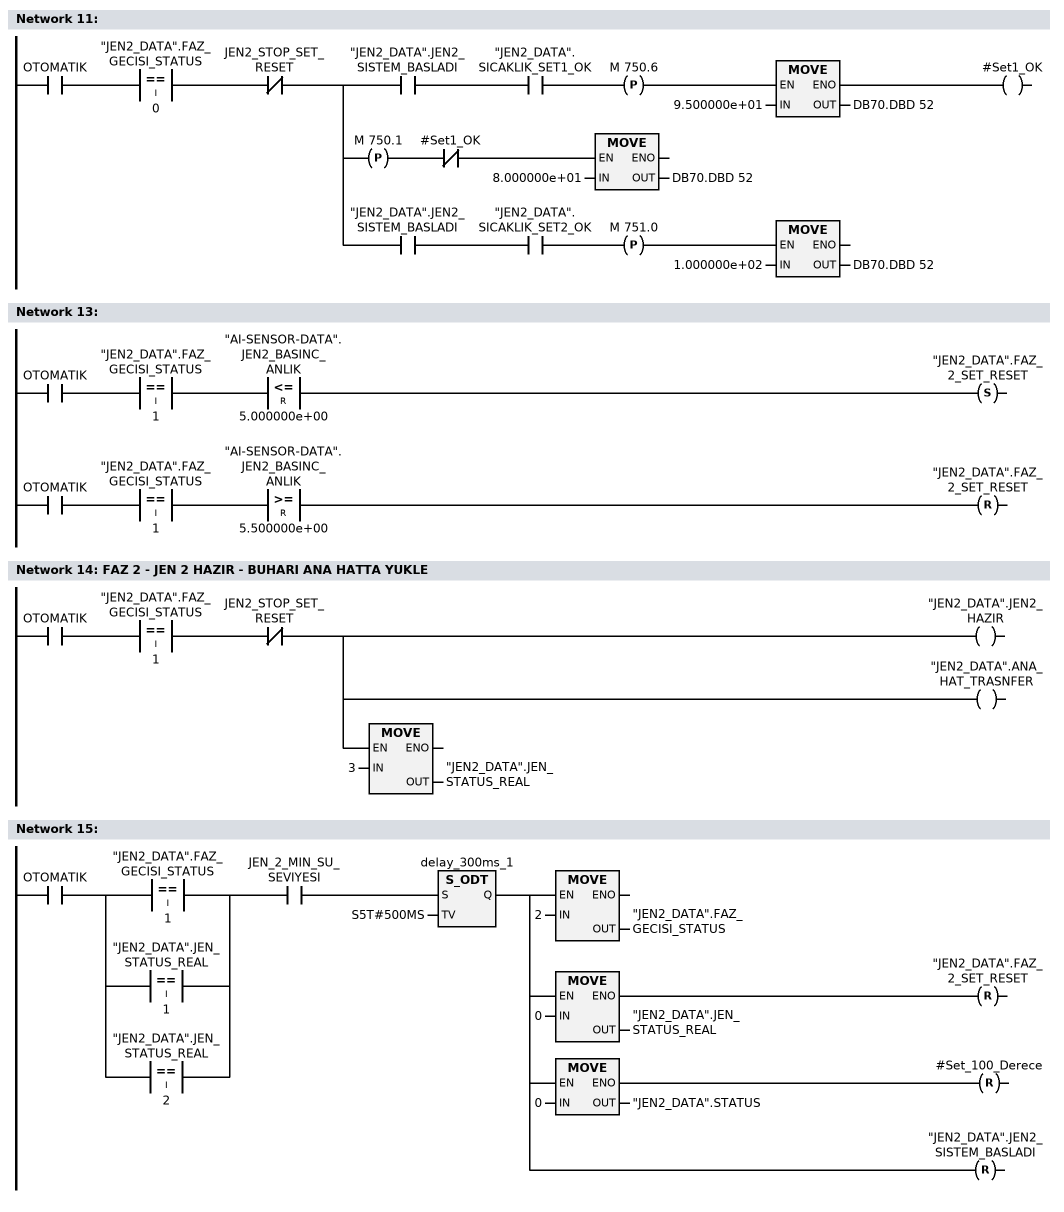
NETWORK
TITLE =
//-Sicaklik set 1 e geldiginde vana kapanma orani 5'e kadar düsüyor
//-Sicaklik set 2 e geldiginde vana kapanma orani 0'a kadar dusecek
      A     "OTOMATIK";
      A(;
      L     "JEN2_DATA".FAZ_GECISI_STATUS;
      L     0;
      ==I;
      );
      AN    "JEN2_STOP_SET_RESET";
      =     L 0.0;
      A     L 0.0;
      A     "JEN2_DATA".JEN2_SISTEM_BASLADI;
      A     "JEN2_DATA".SICAKLIK_SET1_OK;
      FP    M 750.6;
      JNB   _00c;
      L     9.500000e+01;
      T     DB70.DBD 52;
      SET;
      SAVE;
      CLR;
_00c: A     BR;
      =     #Set1_OK;
      A     L 0.0;
      FP    M 750.1;
      AN    #Set1_OK;
      JNB   _00d;
      L     8.000000e+01;
      T     DB70.DBD 52;
_00d: NOP   0;
      A     L 0.0;
      A     "JEN2_DATA".JEN2_SISTEM_BASLADI;
      A     "JEN2_DATA".SICAKLIK_SET2_OK;
      FP    M 751.0;
      JNB   _00e;
      L     1.000000e+02;
      T     DB70.DBD 52;
_00e: NOP   0;
NETWORK
TITLE =
NETWORK
TITLE =
//FAZ - 2 MODUNA GEÇ
//1-BURLOR VE POMPA 4.5-5.5 BAR ARASINDA ÇALISIP DURACAK
      A     "OTOMATIK";
      A(;
      L     "JEN2_DATA".FAZ_GECISI_STATUS;
      L     1;
      ==I;
      );
      A(;
      L     "AI-SENSOR-DATA".JEN2_BASINC_ANLIK;
      L     5.000000e+00;
      <=R;
      );
      S     "JEN2_DATA".FAZ_2_SET_RESET;
      A     "OTOMATIK";
      A(;
      L     "JEN2_DATA".FAZ_GECISI_STATUS;
      L     1;
      ==I;
      );
      A(;
      L     "AI-SENSOR-DATA".JEN2_BASINC_ANLIK;
      L     5.500000e+00;
      >=R;
      );
      R     "JEN2_DATA".FAZ_2_SET_RESET;
      NOP   0;
NETWORK
TITLE = FAZ 2 - JEN 2 HAZIR - BUHARI ANA HATTA YUKLE
      A     "OTOMATIK";
      A(;
      L     "JEN2_DATA".FAZ_GECISI_STATUS;
      L     1;
      ==I;
      );
      AN    "JEN2_STOP_SET_RESET";
      =     L 0.0;
      A     L 0.0;
      BLD   102;
      =     "JEN2_DATA".JEN2_HAZIR;
      A     L 0.0;
      BLD   102;
      =     "JEN2_DATA".ANA_HAT_TRASNFER;
      A     L 0.0;
      JNB   _00f;
      L     3;
      T     "JEN2_DATA".JEN_STATUS_REAL;
_00f: NOP   0;
NETWORK
TITLE =
//FAZ 3 - GUVENLIK ONLEMLERI 
//1- 6 bar asildiginda -ok
//2- Baca 180 dereceyi gecerse -ok
//3- Su miktari min altina duserse -ok
      A     "OTOMATIK";
      A(;
      O(;
      L     "JEN2_DATA".FAZ_GECISI_STATUS;
      L     1;
      ==I;
      );
      O(;
      L     "JEN2_DATA".JEN_STATUS_REAL;
      L     1;
      ==I;
      );
      O(;
      L     "JEN2_DATA".JEN_STATUS_REAL;
      L     2;
      ==I;
      );
      );
      A     "JEN_2_MIN_SU_SEVIYESI";
      L     S5T#500MS;
      SD    "delay_300ms_1";
      NOP   0;
      NOP   0;
      NOP   0;
      A     "delay_300ms_1";
      =     L 0.0;
      A     L 0.0;
      JNB   _010;
      L     2;
      T     "JEN2_DATA".FAZ_GECISI_STATUS;
_010: NOP   0;
      A     L 0.0;
      JNB   _011;
      L     0;
      T     "JEN2_DATA".JEN_STATUS_REAL;
      SET;
      SAVE;
      CLR;
_011: A     BR;
      R     "JEN2_DATA".FAZ_2_SET_RESET;
      A     L 0.0;
      JNB   _012;
      L     0;
      T     "JEN2_DATA".STATUS;
      SET;
      SAVE;
      CLR;
_012: A     BR;
      R     #Set_100_Derece;
      A     L 0.0;
      BLD   102;
      R     "JEN2_DATA".JEN2_SISTEM_BASLADI;
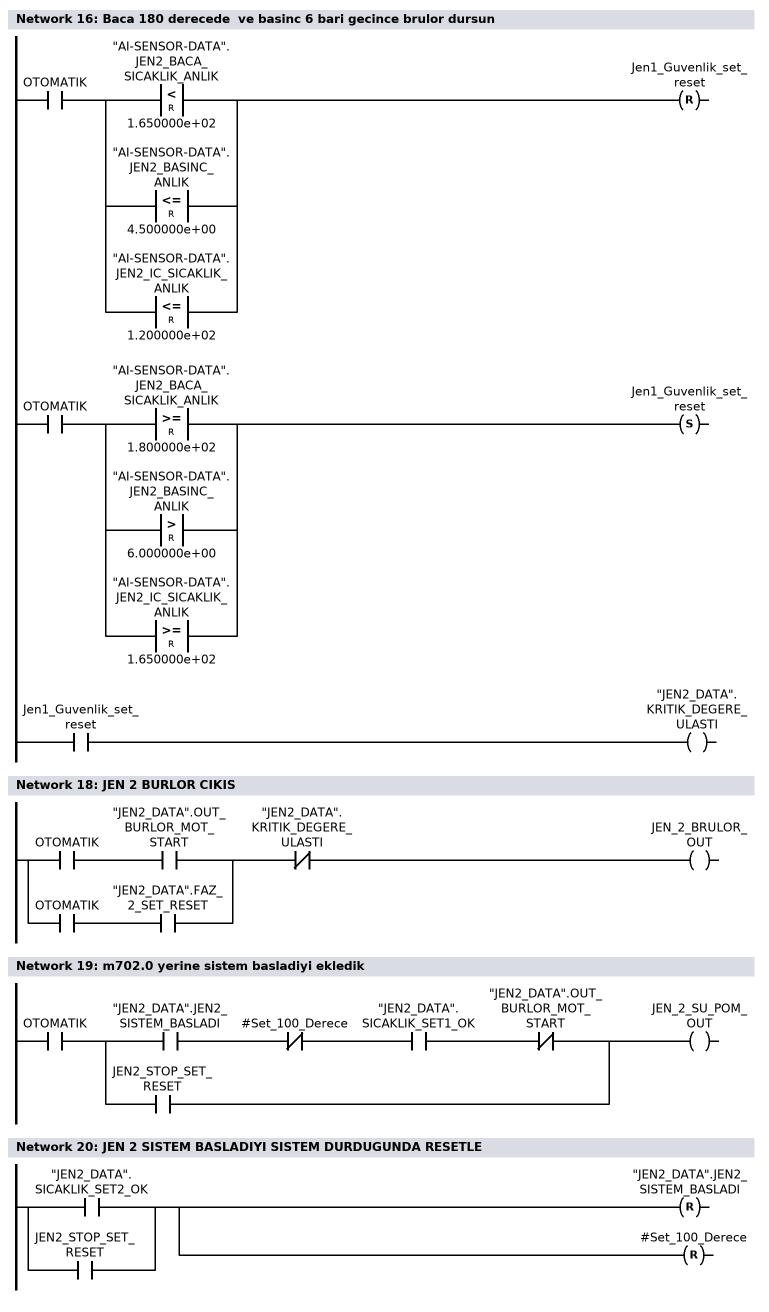
NETWORK
TITLE = Baca 180 derecede  ve basinc 6 bari gecince brulor dursun
      A     "OTOMATIK";
      A(;
      O(;
      L     "AI-SENSOR-DATA".JEN2_BACA_SICAKLIK_ANLIK;
      L     1.650000e+02;
      <R;
      );
      O(;
      L     "AI-SENSOR-DATA".JEN2_BASINC_ANLIK;
      L     4.500000e+00;
      <=R;
      );
      O(;
      L     "AI-SENSOR-DATA".JEN2_IC_SICAKLIK_ANLIK;
      L     1.200000e+02;
      <=R;
      );
      );
      R     "Jen1_Guvenlik_set_reset";
      A     "OTOMATIK";
      A(;
      O(;
      L     "AI-SENSOR-DATA".JEN2_BACA_SICAKLIK_ANLIK;
      L     1.800000e+02;
      >=R;
      );
      O(;
      L     "AI-SENSOR-DATA".JEN2_BASINC_ANLIK;
      L     6.000000e+00;
      >R;
      );
      O(;
      L     "AI-SENSOR-DATA".JEN2_IC_SICAKLIK_ANLIK;
      L     1.650000e+02;
      >=R;
      );
      );
      S     "Jen1_Guvenlik_set_reset";
      A     "Jen1_Guvenlik_set_reset";
      =     "JEN2_DATA".KRITIK_DEGERE_ULASTI;
NETWORK
TITLE =
NETWORK
TITLE = JEN 2 BURLOR CIKIS
      A(;
      A     "OTOMATIK";
      A     "JEN2_DATA".OUT_BURLOR_MOT_START;
      O;
      A     "OTOMATIK";
      A     "JEN2_DATA".FAZ_2_SET_RESET;
      );
      AN    "JEN2_DATA".KRITIK_DEGERE_ULASTI;
      =     "JEN_2_BRULOR_OUT";
NETWORK
TITLE = m702.0 yerine sistem basladiyi ekledik
      A     "OTOMATIK";
      A(;
      A     "JEN2_DATA".JEN2_SISTEM_BASLADI;
      AN    #Set_100_Derece;
      A     "JEN2_DATA".SICAKLIK_SET1_OK;
      AN    "JEN2_DATA".OUT_BURLOR_MOT_START;
      O     "JEN2_STOP_SET_RESET";
      );
      =     "JEN_2_SU_POM_OUT";
NETWORK
TITLE = JEN 2 SISTEM BASLADIYI SISTEM DURDUGUNDA RESETLE
      O     "JEN2_DATA".SICAKLIK_SET2_OK;
      O     "JEN2_STOP_SET_RESET";
      R     "JEN2_DATA".JEN2_SISTEM_BASLADI;
      R     #Set_100_Derece;
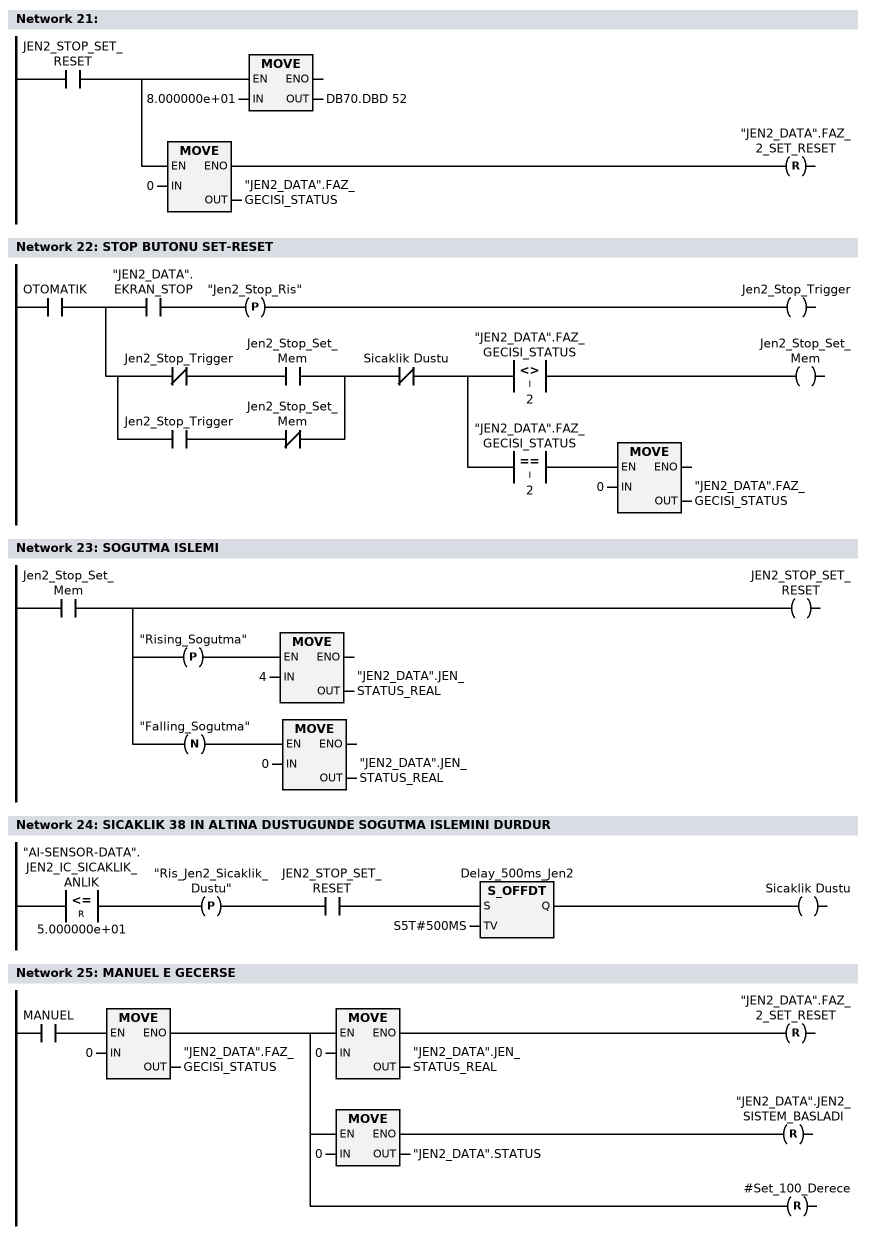
NETWORK
TITLE =
      A     "JEN2_STOP_SET_RESET";
      =     L 0.0;
      A     L 0.0;
      JNB   _013;
      L     8.000000e+01;
      T     DB70.DBD 52;
_013: NOP   0;
      A     L 0.0;
      JNB   _014;
      L     0;
      T     "JEN2_DATA".FAZ_GECISI_STATUS;
      SET;
      SAVE;
      CLR;
_014: A     BR;
      R     "JEN2_DATA".FAZ_2_SET_RESET;
NETWORK
TITLE = STOP BUTONU SET-RESET
      A     "OTOMATIK";
      =     L 0.0;
      A     L 0.0;
      A     "JEN2_DATA".EKRAN_STOP;
      FP    "Jen2_Stop_Ris";
      =     "Jen2_Stop_Trigger";
      A     L 0.0;
      A(;
      AN    "Jen2_Stop_Trigger";
      A     "Jen2_Stop_Set_Mem";
      O;
      A     "Jen2_Stop_Trigger";
      AN    "Jen2_Stop_Set_Mem";
      );
      AN    "Sicaklik Dustu";
      =     L 0.1;
      A     L 0.1;
      A(;
      L     "JEN2_DATA".FAZ_GECISI_STATUS;
      L     2;
      <>I;
      );
      =     "Jen2_Stop_Set_Mem";
      A     L 0.1;
      A(;
      L     "JEN2_DATA".FAZ_GECISI_STATUS;
      L     2;
      ==I;
      );
      JNB   _015;
      L     0;
      T     "JEN2_DATA".FAZ_GECISI_STATUS;
_015: NOP   0;
NETWORK
TITLE = SOGUTMA ISLEMI
      A     "Jen2_Stop_Set_Mem";
      =     L 0.0;
      A     L 0.0;
      BLD   102;
      =     "JEN2_STOP_SET_RESET";
      A     L 0.0;
      FP    "Rising_Sogutma";
      JNB   _016;
      L     4;
      T     "JEN2_DATA".JEN_STATUS_REAL;
_016: NOP   0;
      A     L 0.0;
      FN    "Falling_Sogutma";
      JNB   _017;
      L     0;
      T     "JEN2_DATA".JEN_STATUS_REAL;
_017: NOP   0;
NETWORK
TITLE = SICAKLIK 38 IN ALTINA DUSTUGUNDE SOGUTMA ISLEMINI DURDUR
      A(;
      L     "AI-SENSOR-DATA".JEN2_IC_SICAKLIK_ANLIK;
      L     5.000000e+01;
      <=R;
      );
      FP    "Ris_Jen2_Sicaklik_Dustu";
      A     "JEN2_STOP_SET_RESET";
      L     S5T#500MS;
      SF    "Delay_500ms_Jen2";
      NOP   0;
      NOP   0;
      NOP   0;
      A     "Delay_500ms_Jen2";
      =     "Sicaklik Dustu";
NETWORK
TITLE = MANUEL E GECERSE
      A     "MANUEL";
      JNB   _018;
      L     0;
      T     "JEN2_DATA".FAZ_GECISI_STATUS;
      SET;
      SAVE;
      CLR;
_018: A     BR;
      =     L 0.0;
      A     L 0.0;
      JNB   _019;
      L     0;
      T     "JEN2_DATA".JEN_STATUS_REAL;
      SET;
      SAVE;
      CLR;
_019: A     BR;
      R     "JEN2_DATA".FAZ_2_SET_RESET;
      A     L 0.0;
      JNB   _01a;
      L     0;
      T     "JEN2_DATA".STATUS;
      SET;
      SAVE;
      CLR;
_01a: A     BR;
      R     "JEN2_DATA".JEN2_SISTEM_BASLADI;
      A     L 0.0;
      BLD   102;
      R     #Set_100_Derece;
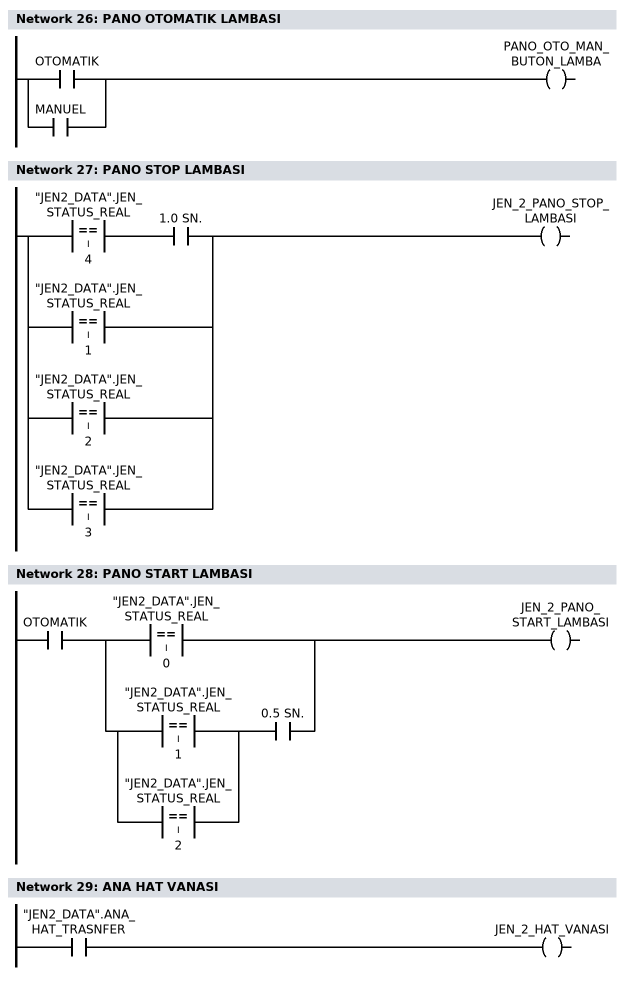
NETWORK
TITLE = PANO OTOMATIK LAMBASI
      O     "OTOMATIK";
      O     "MANUEL";
      =     "PANO_OTO_MAN_BUTON_LAMBA";
NETWORK
TITLE = PANO STOP LAMBASI
//1- Buhar hazýrlaniyor
//2- set 1 e ulasti
//3- Basinci Stabil tutma
//4- Sogutma
      A(;
      L     "JEN2_DATA".JEN_STATUS_REAL;
      L     4;
      ==I;
      );
      A     "1.0 SN.";
      O(;
      L     "JEN2_DATA".JEN_STATUS_REAL;
      L     1;
      ==I;
      );
      O(;
      L     "JEN2_DATA".JEN_STATUS_REAL;
      L     2;
      ==I;
      );
      O(;
      L     "JEN2_DATA".JEN_STATUS_REAL;
      L     3;
      ==I;
      );
      =     "JEN_2_PANO_STOP_LAMBASI";
NETWORK
TITLE = PANO START LAMBASI
      A     "OTOMATIK";
      A(;
      O(;
      L     "JEN2_DATA".JEN_STATUS_REAL;
      L     0;
      ==I;
      );
      O;
      A(;
      O(;
      L     "JEN2_DATA".JEN_STATUS_REAL;
      L     1;
      ==I;
      );
      O(;
      L     "JEN2_DATA".JEN_STATUS_REAL;
      L     2;
      ==I;
      );
      );
      A     "0.5 SN.";
      );
      =     "JEN_2_PANO_START_LAMBASI";
NETWORK
TITLE = ANA HAT VANASI 
      A     "JEN2_DATA".ANA_HAT_TRASNFER;
      =     "JEN_2_HAT_VANASI";
END_FUNCTION_BLOCK

FUNCTION "TIME_UNSCALE" : VOID	// FC 1
VERSION : 0.0
VAR_INPUT
  iTimeET : TIME ;
  iIstenileSure : S5TIME ;
END_VAR
VAR_OUTPUT
  oOUT : DINT ;
END_VAR
VAR_TEMP
  vTemp : DINT ;
  vValue : DINT ;
  vValue2 : DINT ;
  vIstenilenTime : TIME ;
  vIstenilenDint : DINT ;
END_VAR
BEGIN
// body was compiled from an SCL source; compiled code not shown
END_FUNCTION

// FC 33: know-how protected block, not included

// FC 105: know-how protected block, not included

// FC 106: know-how protected block, not included

DATA_BLOCK "AI-SENSOR-DATA"	// DB 1
VERSION : 0.1
  STRUCT
   JEN1_BASINC_ANLIK : REAL ;
   JEN2_BASINC_ANLIK : REAL ;
   JEN1_BASINC_RET_VAL : WORD ;
   JEN2_BASINC_RET_VAL : WORD ;
   JEN1_IC_SICAKLIK_ANLIK : REAL ;
   JEN2_IC_SICAKLIK_ANLIK : REAL ;
   JEN1_IC_SICAKLIK_RET_VAL : WORD ;
   JEN2_IC_SICAKLIK_RET_VAL : WORD ;
   JEN1_BACA_SICAKLIK_ANLIK : REAL ;
   JEN2_BACA_SICAKLIK_ANLIK : REAL ;
   JEN1_BACA_SICAKLIK_RET_V : WORD ;
   JEN2_BACA_SICAKLIK_RET_V : WORD ;
   HAT_BASINCI_RET_V : WORD ;
   HAT_BASINCI_ANLIK : REAL ;
   HAVA_BASINCI_RET_V : WORD ;
   HAVA_BASINCI_ANLIK : REAL ;
   HAT_BASINCI_YETERLI : BOOL ;
  END_STRUCT ;	
BEGIN
END_DATA_BLOCK

DATA_BLOCK "ORTAK_DATA"	// DB 2
VERSION : 0.1
  STRUCT
   JEN_EMNIYET_BASINCI : REAL ;
   JEN_EMNIYET_SICAKLIGI : REAL ;
   OTO_EMNIYET_BASINCI : REAL ;
   OTO_EMNIYET_SICAKLIGI : REAL ;
   OTO_ISLEM_BITTI_VANA_AC : BOOL ;
   OTO_JEN_DURDU : REAL ;
  END_STRUCT ;	
BEGIN
END_DATA_BLOCK

DATA_BLOCK "TIME_OTO_1_DB"	// DB 5
AUTHOR : SIMATIC
FAMILY : IEC_TC
VERSION : 0.0
"TON"
BEGIN
END_DATA_BLOCK

DATA_BLOCK "TIME_OTO_2_DB"	// DB 6
AUTHOR : SIMATIC
FAMILY : IEC_TC
VERSION : 0.0
"TON"
BEGIN
END_DATA_BLOCK

DATA_BLOCK "TIME_OTO_1_PROSES_DB"	// DB 7
AUTHOR : SIMATIC
FAMILY : IEC_TC
VERSION : 0.0
"TON"
BEGIN
END_DATA_BLOCK

DATA_BLOCK "TIME_OTO_2_PROSES_DB"	// DB 8
AUTHOR : SIMATIC
FAMILY : IEC_TC
VERSION : 0.0
"TON"
BEGIN
END_DATA_BLOCK

DATA_BLOCK DB 9
AUTHOR : SIMATIC
FAMILY : IEC_TC
VERSION : 0.0
"TON"
BEGIN
END_DATA_BLOCK

DATA_BLOCK DB 10
AUTHOR : SIMATIC
FAMILY : IEC_TC
VERSION : 0.0
"TON"
BEGIN
END_DATA_BLOCK

DATA_BLOCK "SURELER_DB"	// DB 14
VERSION : 0.0
"SURELER"
BEGIN
END_DATA_BLOCK

DATA_BLOCK "SAFETY_DB"	// DB 15
VERSION : 0.0
"SAFETY"
BEGIN
END_DATA_BLOCK

DATA_BLOCK "KAZAN1_DATA"	// DB 17
VERSION : 0.1
  STRUCT
   IN_STATUS : INT ;
   IN_JEN_OK : BOOL ;
   IN_DIGER_KAZ_TRANS_HAZIR : BOOL ;
   IN_PISIM_SURESI : S5TIME ;
   IN_SCALE_BASINC_PER : INT ;
   IN_SET_BASINC : REAL ;
   IN_DIGER_KAZAN_BASINCI : REAL ;
   O_PID_MAN_ON : BOOL ;
   O_PID_MAN : REAL ;
   O_TRANSFER_YAPILIYOR : BOOL ;
   O_SCALE_BASINC_RET_VAL : WORD ;
   O_SCALE_BASINC_OUT : REAL ;
   O_TRANSFERE_HAZIR : BOOL ;
   O_SCALE_SICAKLIK_RET_VAL : WORD ;
   O_SCALE_SICAKLIK_OUT : REAL ;
   IN_SCALE_SICAKLIK_PER : INT ;
   O_KAZAN_BOSALTIMDA : BOOL ;
   IN_DIGER_KAZ_BOSALTIMDA : BOOL ;
   IN_DIGER_KAZ_TRANSFERDE : BOOL ;
   O_PISIM_BASLADI : BOOL ;
   PISIM_GECEN_SURE_TIME : TIME ;
   PISIM_GECEN_SURE_DINT : DINT ;
   PROSES_SURESI_TIME : TIME ;
   PROSES_SURESI_DINT : DINT ;
   BEKLEME_SURESI_TIME : TIME ;
   BEKLEME_SURESI_DINT : DINT ;
  END_STRUCT ;	
BEGIN
END_DATA_BLOCK

DATA_BLOCK "KAZAN2_DATA"	// DB 18
VERSION : 0.1
  STRUCT
   IN_STATUS : INT ;
   IN_JEN_OK : BOOL ;
   IN_DIGER_KAZ_TRANS_HAZIR : BOOL ;
   IN_PISIM_SURESI : S5TIME ;
   IN_SCALE_BASINC_PER : INT ;
   IN_SET_BASINC : REAL ;
   IN_DIGER_KAZAN_BASINCI : REAL ;
   O_PID_MAN_ON : BOOL ;
   O_PID_MAN : REAL ;
   O_TRANSFER_YAPILIYOR : BOOL ;
   O_SCALE_BASINC_RET_VAL : WORD ;
   O_SCALE_BASINC_OUT : REAL ;
   O_TRANSFERE_HAZIR : BOOL ;
   O_SCALE_SICAKLIK_RET_VAL : WORD ;
   O_SCALE_SICAKLIK_OUT : REAL ;
   IN_SCALE_SICAKLIK_PER : INT ;
   O_KAZAN_BOSALTIMDA : BOOL ;
   IN_DIGER_KAZ_BOSALTIMDA : BOOL ;
   IN_DIGER_KAZ_TRANSFERDE : BOOL ;
   O_PISIM_BASLADI : BOOL ;
   PISIM_GECEN_SURE_TIME : TIME ;
   PISIM_GECEN_SURE_DINT : DINT ;
   PROSES_SURESI_TIM : TIME ;
   PROSES_SURESI_DINT : DINT ;
   BEKLEME_SURESI_TIME : TIME ;
   BEKLEME_SURESI_DINT : DINT ;
  END_STRUCT ;	
BEGIN
END_DATA_BLOCK

DATA_BLOCK "JEN1_DATA"	// DB 19
VERSION : 0.1
  STRUCT
   BASINC_SET_POINT : REAL ;
   STATUS : INT ;
   SICAKLIK_SET_POINT_1 : REAL ;
   SICAKLIK_SET_POINT_2 : REAL ;
   SISTEM_BASLADI : BOOL ;
   EKRAN_START : BOOL ;
   EKRAN_STOP : BOOL ;
   OUT_BURLOR_MOT_START : BOOL ;
   SICAKLIK_SET1_OK : BOOL ;
   SICAKLIK_SET2_OK : BOOL ;
   OUT_PID_START : BOOL ;
   FAZ_GECISI_STATUS : INT ;
   FAZ_2_SET_RESET : BOOL ;
   BAR_5_E_ULASTI : BOOL ;
   JEN1_HAZIR : BOOL ;
   ANA_HAT_TRASFER_HAZIR : BOOL ;
   JEN_STATUS_REAL : INT ;
   STOP_SET_RESET : BOOL ;
   CALISMA_SURESI_TIME : TIME ;
   CALISMA_SURESI_DINT : DINT ;
   KRITIK_DEGERLERE_ULASTI : BOOL ;	//180 derece baca-6 bari gecti- 165 ic sicaklik
   CALISMA_SURESI_EKRAN : DINT ;
   SET2_DEGERINE_ULASMADI : BOOL ;
  END_STRUCT ;	
BEGIN
END_DATA_BLOCK

DATA_BLOCK "JEN2_DATA"	// DB 20
VERSION : 0.1
  STRUCT
   BASINC_SET_POINT : REAL ;
   STATUS : INT ;
   SICAKLIK_SET_POINT_1 : REAL ;
   SICAKLIK_SET_POINT_2 : REAL ;
   JEN2_SISTEM_BASLADI : BOOL ;
   EKRAN_START : BOOL ;
   EKRAN_STOP : BOOL ;
   OUT_BURLOR_MOT_START : BOOL ;
   SICAKLIK_SET1_OK : BOOL ;
   SICAKLIK_SET2_OK : BOOL ;
   OUT_PID_START : BOOL ;
   FAZ_GECISI_STATUS : INT ;
   FAZ_2_SET_RESET : BOOL ;
   BAR_5_E_ULASTI : BOOL ;
   JEN2_HAZIR : BOOL ;
   ANA_HAT_TRASNFER : BOOL ;
   JEN_STATUS_REAL : INT ;
   STOP_SET_RESET : BOOL ;
   CALISMA_SURESI_TIME : TIME ;
   CALISMA_SURESI_DINT : DINT ;
   KRITIK_DEGERE_ULASTI : BOOL ;	//Baca 180 derecede-6 bari gecti-165 ic sicaklik
   CALISMA_SURESI_EKRAN : DINT ;
  END_STRUCT ;	
BEGIN
END_DATA_BLOCK

DATA_BLOCK "JEN1_PID_DATA"	// DB 21
VERSION : 0.1
  STRUCT
   TCONT_C_LMN : REAL ;
   TCONT_C_LMN_PER : INT ;
  END_STRUCT ;	
BEGIN
END_DATA_BLOCK

DATA_BLOCK "JEN2_PID_DATA"	// DB 22
VERSION : 0.1
  STRUCT
   TCONT_C_LMN : REAL ;
   TCONT_C_LMN_PER : INT ;
  END_STRUCT ;	
BEGIN
END_DATA_BLOCK

DATA_BLOCK "KAZAN1_PID_DATA"	// DB 23
VERSION : 0.1
  STRUCT
   TCONT_LMN_PER : INT ;
   TCONT_LMN : REAL ;
  END_STRUCT ;	
BEGIN
END_DATA_BLOCK

DATA_BLOCK "KAZAN2_PID_DATA"	// DB 24
VERSION : 0.1
  STRUCT
   TCONT_LMN_PER : INT ;
   TCONT_LMN : REAL ;
  END_STRUCT ;	
BEGIN
END_DATA_BLOCK

DATA_BLOCK DB 50
AUTHOR : SIMATIC
FAMILY : ICONT
VERSION : 0.0
"CONT_C"
BEGIN
END_DATA_BLOCK

DATA_BLOCK "JEN2_KONTROL_BLOGU_DB"	// DB 51
VERSION : 0.0
"JEN2_PID_KONTROL"
BEGIN
END_DATA_BLOCK

DATA_BLOCK DB 52
VERSION : 0.0
"JEN1_PID_KONTROL"
BEGIN
END_DATA_BLOCK

DATA_BLOCK "JEN_1_PID_DB"	// DB 69
AUTHOR : SIMATIC
FAMILY : CONTROL
VERSION : 0.0
"TCONT_CP"
BEGIN
END_DATA_BLOCK

DATA_BLOCK "JEN_2_PID_DB"	// DB 70
AUTHOR : SIMATIC
FAMILY : CONTROL
VERSION : 0.0
"TCONT_CP"
BEGIN
END_DATA_BLOCK

DATA_BLOCK "OTOKLAV_1_DB"	// DB 94
VERSION : 0.0
"KAZAN_1_KONTROL"
BEGIN
END_DATA_BLOCK

DATA_BLOCK "OTOKLAV_2_DB"	// DB 95
VERSION : 0.0
"KAZAN_2_KONTROL"
BEGIN
END_DATA_BLOCK

DATA_BLOCK "FB98_DB"	// DB 98
VERSION : 0.0
"JEN1_KONTROL_BLOGU"
BEGIN
END_DATA_BLOCK

DATA_BLOCK "FB99_DB"	// DB 99
VERSION : 0.0
"JEN2_KONTROL_BLOGU"
BEGIN
END_DATA_BLOCK

DATA_BLOCK DB 120
VERSION : 0.0
"KAZAN_ORTAK"
BEGIN
END_DATA_BLOCK

DATA_BLOCK "KAZAN_1_PID_DB"	// DB 130
AUTHOR : SIMATIC
FAMILY : CONTROL
VERSION : 0.0
"TCONT_CP"
BEGIN
END_DATA_BLOCK

DATA_BLOCK DB 131
VERSION : 0.0
"KAZAN_1_PID_KONTROL"
BEGIN
END_DATA_BLOCK

DATA_BLOCK DB 132
VERSION : 0.0
"KAZAN_2_PID_KONTROL"
BEGIN
END_DATA_BLOCK

DATA_BLOCK DB 230
VERSION : 0.0
"KAZAN_ORTAK"
BEGIN
END_DATA_BLOCK

DATA_BLOCK "KAZAN_2_PID_DATA"	// DB 231
AUTHOR : SIMATIC
FAMILY : CONTROL
VERSION : 0.0
"TCONT_CP"
BEGIN
END_DATA_BLOCK

DATA_BLOCK DB 232
VERSION : 0.0
"TEST_BLOGU"
BEGIN
END_DATA_BLOCK

ORGANIZATION_BLOCK OB 1
TITLE = "Main Program Sweep (Cycle)"
VERSION : 0.1
VAR_TEMP
  OB1_EV_CLASS : BYTE ;	//Bits 0-3 = 1 (Coming event), Bits 4-7 = 1 (Event class 1)
  OB1_SCAN_1 : BYTE ;	//1 (Cold restart scan 1 of OB 1), 3 (Scan 2-n of OB 1)
  OB1_PRIORITY : BYTE ;	//Priority of OB Execution
  OB1_OB_NUMBR : BYTE ;	//1 (Organization block 1, OB1)
  OB1_RESERVED_1 : BYTE ;	//Reserved for system
  OB1_RESERVED_2 : BYTE ;	//Reserved for system
  OB1_PREV_CYCLE : INT ;	//Cycle time of previous OB1 scan (milliseconds)
  OB1_MIN_CYCLE : INT ;	//Minimum cycle time of OB1 (milliseconds)
  OB1_MAX_CYCLE : INT ;	//Maximum cycle time of OB1 (milliseconds)
  OB1_DATE_TIME : DATE_AND_TIME ;	//Date and time OB1 started
END_VAR
BEGIN
NETWORK
TITLE = ALWAYS OFF
      UC    "MAINBLOCK";
NETWORK
TITLE = HAVA VE HAT BASINCI
      CALL  "SCALE" (
           $1                       := P#P 292.0,
           $2                       := L#1092616192,
           $3                       := L#0,
           $4                       := "ALWAYS OFF",
           $5                       := "AI-SENSOR-DATA".HAT_BASINCI_RET_V,
           $6                       := "AI-SENSOR-DATA".HAT_BASINCI_ANLIK);
      CALL  "SCALE" (
           $1                       := P#P 294.0,
           $2                       := L#1092616192,
           $3                       := L#0,
           $4                       := "ALWAYS OFF",
           $5                       := "AI-SENSOR-DATA".HAVA_BASINCI_RET_V,
           $6                       := "AI-SENSOR-DATA".HAVA_BASINCI_ANLIK);
NETWORK
TITLE = ACIKLAMALAR
//FB98 - JEN 1 KONTROL BLOGU
//FB99 - JEN 2 KONTROL BLOGU
//FB49 - JEN 1 PID KONTROL - PID BLOKLARI
//FB50 - JEN 2 PID KONTROL - PID BLOKLARI
//FB94 - KAZAN 1 KONTROL BLOGU - KAZAN 1 ILE ILGILI KONTROLLER
//FB95 - KAZAN 2 KONTROL BLOGU - KAZAN 2 ILE ILGILI KONTROLLER
//FB47 - KAZAN 1 PID KONTROL
//FB48 - KAZAN 2 PID KONTROL
//FB3 - SURELER - KAZAN1,KAZAN2, JEN1, JEN2 ILE ILGILI TUM SURELER BURADA TUTULUR
//FB2 - SAFETY
//      1)JEN1, JEN2 KRITIK SU SEVIYE MIKTARLARI
//      2)HAVA BASINCI KONTROLU
//      3)JENERATOR IS BITIMINDE BORUDA KALAN BUHARIN TAHLIYESI
//FB1 - MAINBLOCK  
//      1)ÇALISACAK TUM BLOKLAR BURADA CAGRILIR
//      2)AYRICA HAVA VE HAT BASINCI DONUSUMLARI BURADADIR
//FB5 - TEST BLOGU - PROSESIN DEVREYE ALINAMADAN ONCEKI TEST ISLEMLERININ GERCEKLESTIGI
//      BLOKTUR.
END_ORGANIZATION_BLOCK

ORGANIZATION_BLOCK "PID BLOCK"	// OB 35
TITLE = "Cyclic Interrupt"
VERSION : 0.1
VAR_TEMP
  OB35_EV_CLASS : BYTE ;	//Bits 0-3 = 1 (Coming event), Bits 4-7 = 1 (Event class 1)
  OB35_STRT_INF : BYTE ;	//16#36 (OB 35 has started)
  OB35_PRIORITY : BYTE ;	//Priority of OB Execution
  OB35_OB_NUMBR : BYTE ;	//35 (Organization block 35, OB35)
  OB35_RESERVED_1 : BYTE ;	//Reserved for system
  OB35_RESERVED_2 : BYTE ;	//Reserved for system
  OB35_PHASE_OFFSET : WORD ;	//Phase offset (msec)
  OB35_RESERVED_3 : INT ;	//Reserved for system
  OB35_EXC_FREQ : INT ;	//Frequency of execution (msec)
  OB35_DATE_TIME : DATE_AND_TIME ;	//Date and time OB35 started
END_VAR
BEGIN
NETWORK
TITLE =
      CALL  "JEN1_PID_KONTROL" , DB 52;
      CALL  "JEN2_PID_KONTROL" , "JEN2_KONTROL_BLOGU_DB";
NETWORK
TITLE =
      CALL  "KAZAN_1_PID_KONTROL" , DB 131;
      CALL  "KAZAN_2_PID_KONTROL" , DB 132;
END_ORGANIZATION_BLOCK

ORGANIZATION_BLOCK "ZAMANHATASI"	// OB 80
TITLE = "Cycle Time Fault"
VERSION : 0.1
VAR_TEMP
  OB80_EV_CLASS : BYTE ;	//16#35, Event class 3, Entering event state, Internal fault event
  OB80_FLT_ID : BYTE ;	//16#XX, Fault identifcation code
  OB80_PRIORITY : BYTE ;	//Priority of OB Execution
  OB80_OB_NUMBR : BYTE ;	//80 (Organization block 80, OB80)
  OB80_RESERVED_1 : BYTE ;	//Reserved for system
  OB80_RESERVED_2 : BYTE ;	//Reserved for system
  OB80_ERROR_INFO : WORD ;	//Error information on event
  OB80_ERR_EV_CLASS : BYTE ;	//Class of event causing error
  OB80_ERR_EV_NUM : BYTE ;	//Number of event causing error
  OB80_OB_PRIORITY : BYTE ;	//Priority of OB causing error
  OB80_OB_NUM : BYTE ;	//Number of OB causing error
  OB80_DATE_TIME : DATE_AND_TIME ;	//Date and time OB80 started
END_VAR
BEGIN
// (block stored without names or comments; labels and parameter names are numbered)
END_ORGANIZATION_BLOCK

ORGANIZATION_BLOCK "GERILIMHATASI"	// OB 81
TITLE = "Power Supply Fault"
VERSION : 0.1
VAR_TEMP
  OB81_EV_CLASS : BYTE ;	//16#39, Event class 3, Entering event state, Internal fault event
  OB81_FLT_ID : BYTE ;	//16#XX, Fault identifcation code
  OB81_PRIORITY : BYTE ;	//Priority of OB Execution
  OB81_OB_NUMBR : BYTE ;	//81 (Organization block 81, OB81)
  OB81_RESERVED_1 : BYTE ;	//Reserved for system
  OB81_RESERVED_2 : BYTE ;	//Reserved for system
  OB81_RACK_CPU : WORD ;	//see online help (F1)
  OB81_RESERVED_3 : BYTE ;	//Reserved for system
  OB81_RESERVED_4 : BYTE ;	//Reserved for system
  OB81_RESERVED_5 : BYTE ;	//Reserved for system
  OB81_RESERVED_6 : BYTE ;	//Reserved for system
  OB81_DATE_TIME : DATE_AND_TIME ;	//Date and time OB81 started
END_VAR
BEGIN
// (block stored without names or comments; labels and parameter names are numbered)
END_ORGANIZATION_BLOCK

ORGANIZATION_BLOCK "HATAUYARISI"	// OB 82
TITLE = "I/O Point Fault"
VERSION : 0.1
VAR_TEMP
  OB82_EV_CLASS : BYTE ;	//16#39, Event class 3, Entering event state, Internal fault event
  OB82_FLT_ID : BYTE ;	//16#XX, Fault identifcation code
  OB82_PRIORITY : BYTE ;	//Priority of OB Execution
  OB82_OB_NUMBR : BYTE ;	//82 (Organization block 82, OB82)
  OB82_RESERVED_1 : BYTE ;	//Reserved for system
  OB82_IO_FLAG : BYTE ;	//Input (01010100), Output (01010101)
  OB82_MDL_ADDR : WORD ;	//Base address of module with fault
  OB82_MDL_DEFECT : BOOL ;	//Module defective
  OB82_INT_FAULT : BOOL ;	//Internal fault
  OB82_EXT_FAULT : BOOL ;	//External fault
  OB82_PNT_INFO : BOOL ;	//Point information
  OB82_EXT_VOLTAGE : BOOL ;	//External voltage low
  OB82_FLD_CONNCTR : BOOL ;	//Field wiring connector missing
  OB82_NO_CONFIG : BOOL ;	//Module has no configuration data
  OB82_CONFIG_ERR : BOOL ;	//Module has configuration error
  OB82_MDL_TYPE : BYTE ;	//Type of module
  OB82_SUB_MDL_ERR : BOOL ;	//Sub-Module is missing or has error
  OB82_COMM_FAULT : BOOL ;	//Communication fault
  OB82_MDL_STOP : BOOL ;	//Module is stopped
  OB82_WTCH_DOG_FLT : BOOL ;	//Watch dog timer stopped module
  OB82_INT_PS_FLT : BOOL ;	//Internal power supply fault
  OB82_PRIM_BATT_FLT : BOOL ;	//Primary battery is in fault
  OB82_BCKUP_BATT_FLT : BOOL ;	//Backup battery is in fault
  OB82_RESERVED_2 : BOOL ;	//Reserved for system
  OB82_RACK_FLT : BOOL ;	//Rack fault, only for bus interface module
  OB82_PROC_FLT : BOOL ;	//Processor fault
  OB82_EPROM_FLT : BOOL ;	//EPROM fault
  OB82_RAM_FLT : BOOL ;	//RAM fault
  OB82_ADU_FLT : BOOL ;	//ADU fault
  OB82_FUSE_FLT : BOOL ;	//Fuse fault
  OB82_HW_INTR_FLT : BOOL ;	//Hardware interupt input in fault
  OB82_RESERVED_3 : BOOL ;	//Reserved for system
  OB82_DATE_TIME : DATE_AND_TIME ;	//Date and time OB82 started
END_VAR
BEGIN
// (block stored without names or comments; labels and parameter names are numbered)
END_ORGANIZATION_BLOCK

ORGANIZATION_BLOCK "TAKMACIKARMAHATASI"	// OB 83
TITLE = "I/O Point Fault"
VERSION : 0.1
VAR_TEMP
  OB83_EV_CLASS : BYTE ;	//16#38/39, Event class 3, module inserted/removed (8/9)
  OB83_FLT_ID : BYTE ;	//16#XX, Fault identifcation code
  OB83_PRIORITY : BYTE ;	//Priority of OB Execution
  OB83_OB_NUMBR : BYTE ;	//83 (Organization block 83, OB83)
  OB83_RESERVED_1 : BYTE ;	//Reserved for system
  OB83_MDL_ID : BYTE ;	//Input module (01010100), Output module (01010101)
  OB83_MDL_ADDR : WORD ;	//Base address of module with point fault
  OB83_RACK_NUM : INT ;	//Number of rack that has module with point fault
  OB83_MDL_TYPE : WORD ;	//Module type with point fault
  OB83_DATE_TIME : DATE_AND_TIME ;	//Date and time OB83 started
END_VAR
BEGIN
// (block stored without names or comments; labels and parameter names are numbered)
END_ORGANIZATION_BLOCK

ORGANIZATION_BLOCK "CPUHARDWAREERROR"	// OB 84
TITLE = "CPU Fault"
VERSION : 0.1
VAR_TEMP
  OB84_EV_CLASS : BYTE ;	//16#38/39, Event class 3, module inserted/removed (8/9)
  OB84_FLT_ID : BYTE ;	//16#81, Fault identifcation code
  OB84_PRIORITY : BYTE ;	//Priority of OB Execution
  OB84_OB_NUMBR : BYTE ;	//84 (Organization block 84, OB84)
  OB84_RESERVED_1 : BYTE ;	//Reserved for system
  OB84_RESERVED_2 : BYTE ;	//Reserved for system
  OB84_RESERVED_3 : WORD ;	//Reserved for system
  OB84_RESERVED_4 : DWORD ;	//Reserved for system
  OB84_DATE_TIME : DATE_AND_TIME ;	//Date and time OB84 started
END_VAR
BEGIN
// (block stored without names or comments; labels and parameter names are numbered)
END_ORGANIZATION_BLOCK

ORGANIZATION_BLOCK "PROGRAMHATASI"	// OB 85
TITLE = "Organization Block (OB) Not Loaded Fault"
VERSION : 0.1
VAR_TEMP
  OB85_EV_CLASS : BYTE ;	//16#35 Event class 3
  OB85_FLT_ID : BYTE ;	//16#XX, Fault identification code
  OB85_PRIORITY : BYTE ;	//Priority of OB Execution
  OB85_OB_NUMBR : BYTE ;	//85 (Organization block 85, OB85)
  OB85_RESERVED_1 : BYTE ;	//Reserved for system
  OB85_RESERVED_2 : BYTE ;	//Reserved for system
  OB85_RESERVED_3 : INT ;	//Reserved for system
  OB85_ERR_EV_CLASS : BYTE ;	//Class of event causing error
  OB85_ERR_EV_NUM : BYTE ;	//Number of event causing error
  OB85_OB_PRIOR : BYTE ;	//Priority of OB causing error
  OB85_OB_NUM : BYTE ;	//Number of OB causing error
  OB85_DATE_TIME : DATE_AND_TIME ;	//Date and time OB85 started
END_VAR
BEGIN
// (block stored without names or comments; labels and parameter names are numbered)
END_ORGANIZATION_BLOCK

ORGANIZATION_BLOCK "RACKHATASI"	// OB 86
TITLE = "Loss Of Rack Fault"
VERSION : 0.1
VAR_TEMP
  OB86_EV_CLASS : BYTE ;	//16#38/39 Event class 3
  OB86_FLT_ID : BYTE ;	//16#C1/C4/C5, Fault identifcation code
  OB86_PRIORITY : BYTE ;	//Priority of OB Execution
  OB86_OB_NUMBR : BYTE ;	//86 (Organization block 86, OB86)
  OB86_RESERVED_1 : BYTE ;	//Reserved for system
  OB86_RESERVED_2 : BYTE ;	//Reserved for system
  OB86_MDL_ADDR : WORD ;	//Base address of IM module in rack with fault
  OB86_RACKS_FLTD : ARRAY  [0 .. 31 ] OF BOOL ;	//Racks in fault
  OB86_DATE_TIME : DATE_AND_TIME ;	//Date and time OB86 started
END_VAR
BEGIN
// (block stored without names or comments; labels and parameter names are numbered)
END_ORGANIZATION_BLOCK

ORGANIZATION_BLOCK "HABERLESMEHATASI"	// OB 87
TITLE = "Communication Fault"
VERSION : 0.1
VAR_TEMP
  OB87_EV_CLASS : BYTE ;	//16#39 Event class 3
  OB87_FLT_ID : BYTE ;	//16#XX, Fault identifcation code
  OB87_PRIORITY : BYTE ;	//Priority of OB Execution
  OB87_OB_NUMBR : BYTE ;	//87 (Organization block 87, OB87)
  OB87_RESERVED_1 : BYTE ;	//Reserved for system
  OB87_RESERVED_2 : BYTE ;	//Reserved for system
  OB87_RESERVED_3 : WORD ;	//Reserved for system
  OB87_RESERVED_4 : DWORD ;	//Reserved for system
  OB87_DATE_TIME : DATE_AND_TIME ;	//Date and time OB87 started
END_VAR
BEGIN
// (block stored without names or comments; labels and parameter names are numbered)
END_ORGANIZATION_BLOCK

ORGANIZATION_BLOCK "COMPLETE RESTART"	// OB 100
TITLE = "Complete Restart"
VERSION : 0.1
VAR_TEMP
  OB100_EV_CLASS : BYTE ;	//16#13, Event class 1, Entering event state, Event logged in diagnostic buffer
  OB100_STRTUP : BYTE ;	//16#81/82/83/84 Method of startup
  OB100_PRIORITY : BYTE ;	//Priority of OB Execution
  OB100_OB_NUMBR : BYTE ;	//100 (Organization block 100, OB100)
  OB100_RESERVED_1 : BYTE ;	//Reserved for system
  OB100_RESERVED_2 : BYTE ;	//Reserved for system
  OB100_STOP : WORD ;	//Event that caused CPU to stop (16#4xxx)
  OB100_STRT_INFO : DWORD ;	//Information on how system started
  OB100_DATE_TIME : DATE_AND_TIME ;	//Date and time OB100 started
END_VAR
BEGIN
NETWORK
TITLE = Kazan islemlerini sifirlama islemleri
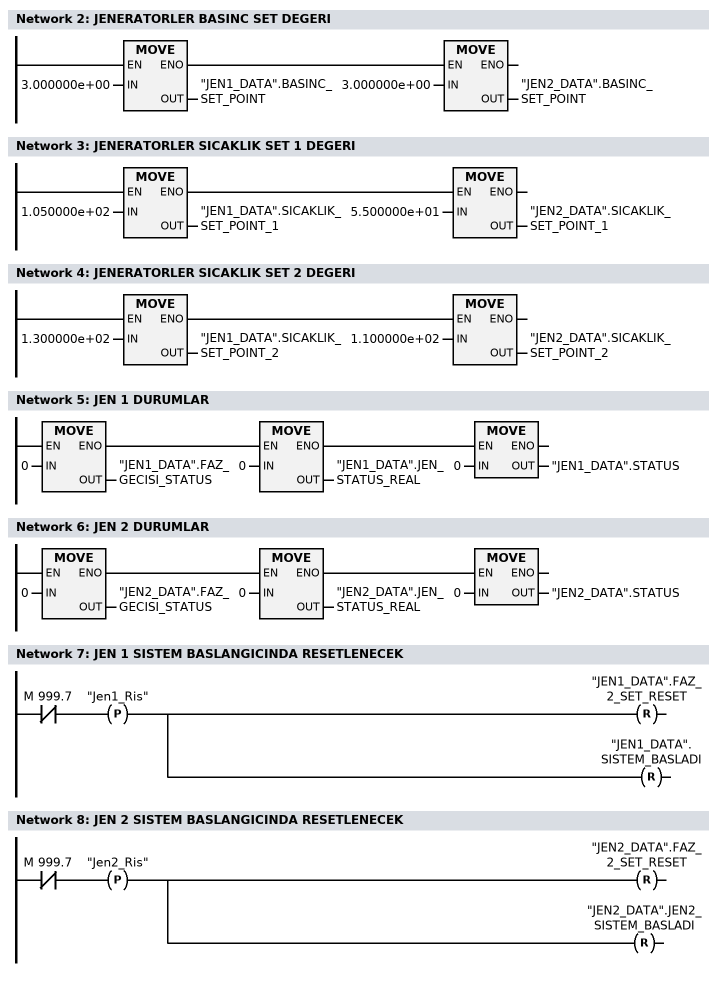
NETWORK
TITLE = JENERATORLER BASINC SET DEGERI
      A(;
      L     3.000000e+00;
      T     "JEN1_DATA".BASINC_SET_POINT;
      SET;
      SAVE;
      CLR;
      A     BR;
      );
      JNB   _001;
      L     3.000000e+00;
      T     "JEN2_DATA".BASINC_SET_POINT;
_001: NOP   0;
NETWORK
TITLE = JENERATORLER SICAKLIK SET 1 DEGERI
      A(;
      L     1.050000e+02;
      T     "JEN1_DATA".SICAKLIK_SET_POINT_1;
      SET;
      SAVE;
      CLR;
      A     BR;
      );
      JNB   _002;
      L     5.500000e+01;
      T     "JEN2_DATA".SICAKLIK_SET_POINT_1;
_002: NOP   0;
NETWORK
TITLE = JENERATORLER SICAKLIK SET 2 DEGERI
      A(;
      L     1.300000e+02;
      T     "JEN1_DATA".SICAKLIK_SET_POINT_2;
      SET;
      SAVE;
      CLR;
      A     BR;
      );
      JNB   _003;
      L     1.100000e+02;
      T     "JEN2_DATA".SICAKLIK_SET_POINT_2;
_003: NOP   0;
NETWORK
TITLE = JEN 1 DURUMLAR
      A(;
      A(;
      L     0;
      T     "JEN1_DATA".FAZ_GECISI_STATUS;
      SET;
      SAVE;
      CLR;
      A     BR;
      );
      JNB   _004;
      L     0;
      T     "JEN1_DATA".JEN_STATUS_REAL;
      SET;
      SAVE;
      CLR;
_004: A     BR;
      );
      JNB   _005;
      L     0;
      T     "JEN1_DATA".STATUS;
_005: NOP   0;
NETWORK
TITLE = JEN 2 DURUMLAR
      A(;
      A(;
      L     0;
      T     "JEN2_DATA".FAZ_GECISI_STATUS;
      SET;
      SAVE;
      CLR;
      A     BR;
      );
      JNB   _006;
      L     0;
      T     "JEN2_DATA".JEN_STATUS_REAL;
      SET;
      SAVE;
      CLR;
_006: A     BR;
      );
      JNB   _007;
      L     0;
      T     "JEN2_DATA".STATUS;
_007: NOP   0;
NETWORK
TITLE = JEN 1 SISTEM BASLANGICINDA RESETLENECEK
      AN    M 999.7;
      FP    "Jen1_Ris";
      R     "JEN1_DATA".FAZ_2_SET_RESET;
      R     "JEN1_DATA".SISTEM_BASLADI;
NETWORK
TITLE = JEN 2 SISTEM BASLANGICINDA RESETLENECEK
      AN    M 999.7;
      FP    "Jen2_Ris";
      R     "JEN2_DATA".FAZ_2_SET_RESET;
      R     "JEN2_DATA".JEN2_SISTEM_BASLADI;
END_ORGANIZATION_BLOCK

ORGANIZATION_BLOCK "RESTART"	// OB 101
TITLE = "Restart"
VERSION : 0.1
VAR_TEMP
  OB101_EV_CLASS : BYTE ;	//16#13, Event class 1, Entering event state, Event logged in diagnostic buffer
  OB101_STRTUP : BYTE ;	//16#81/82/83/84 Method of startup
  OB101_PRIORITY : BYTE ;	//Priority of OB Execution
  OB101_OB_NUMBR : BYTE ;	//101 (Organization block 101, OB101)
  OB101_RESERVED_1 : BYTE ;	//Reserved for system
  OB101_RESERVED_2 : BYTE ;	//Reserved for system
  OB101_STOP : WORD ;	//Event that caused CPU to stop (16#4xxx)
  OB101_STRT_INFO : DWORD ;	//Information on how system started
  OB101_DATE_TIME : DATE_AND_TIME ;	//Date and time OB101 started
END_VAR
BEGIN
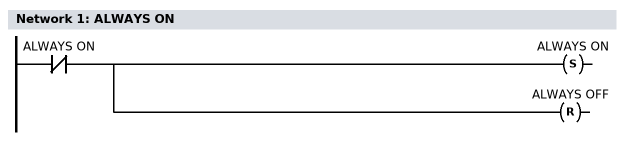
NETWORK
TITLE = ALWAYS ON
      AN    "ALWAYS ON";
      S     "ALWAYS ON";
      R     "ALWAYS OFF";
END_ORGANIZATION_BLOCK

ORGANIZATION_BLOCK "COLD RESTART"	// OB 102
TITLE = "Cold Restart"
VERSION : 0.1
VAR_TEMP
  OB102_EV_CLASS : BYTE ;	//16#13, Event class 1, Entering event state, Event logged in diagnostic buffer
  OB102_STRTUP : BYTE ;	//16#85...8B Method of startup
  OB102_PRIORITY : BYTE ;	//Priority of OB Execution
  OB102_OB_NUMBR : BYTE ;	//102 (Organization block 102, OB102)
  OB102_RESERVED_1 : BYTE ;	//Reserved for system
  OB102_RESERVED_2 : BYTE ;	//Reserved for system
  OB102_STOP : WORD ;	//Event that caused CPU to stop (16#4xxx)
  OB102_STRT_INFO : DWORD ;	//Information on how system started
  OB102_DATE_TIME : DATE_AND_TIME ;	//Date and time OB102 started
END_VAR
BEGIN
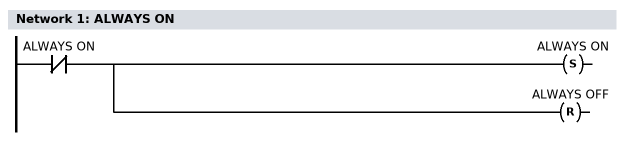
NETWORK
TITLE = ALWAYS ON
      AN    "ALWAYS ON";
      S     "ALWAYS ON";
      R     "ALWAYS OFF";
END_ORGANIZATION_BLOCK

ORGANIZATION_BLOCK "PROGRAMMINGERROR"	// OB 121
TITLE = "Programming Error"
VERSION : 0.1
VAR_TEMP
  OB121_EV_CLASS : BYTE ;	//16#25, Event class 2, Entering event state, Internal fault event
  OB121_SW_FLT : BYTE ;	//16#XX Software programming fault
  OB121_PRIORITY : BYTE ;	//Priority of OB Execution
  OB121_OB_NUMBR : BYTE ;	//121 (Organization block 121, OB121)
  OB121_BLK_TYPE : BYTE ;	//16#88/8A/8B/8C/8E Type of block fault occured in
  OB121_RESERVED_1 : BYTE ;	//Reserved for system
  OB121_FLT_REG : WORD ;	//16#XX Specific register that caused fault
  OB121_BLK_NUM : WORD ;	//Number of block that programming fault occured in
  OB121_PRG_ADDR : WORD ;	//Address in block where programming fault occured
  OB121_DATE_TIME : DATE_AND_TIME ;	//Date and time OB121 started
END_VAR
BEGIN
// (block stored without names or comments; labels and parameter names are numbered)
END_ORGANIZATION_BLOCK

ORGANIZATION_BLOCK "MOD_ERR"	// OB 122
TITLE = "Module Access Error"
VERSION : 0.1
VAR_TEMP
  OB122_EV_CLASS : BYTE ;	//16#29, Event class 2, Entering event state, Internal fault event
  OB122_SW_FLT : BYTE ;	//16#XX Software error code
  OB122_PRIORITY : BYTE ;	//Priority of OB Execution
  OB122_OB_NUMBR : BYTE ;	//122 (Organization block 122, OB122)
  OB122_BLK_TYPE : BYTE ;	//16#88/8C/8E Type of block fault occured in
  OB122_MEM_AREA : BYTE ;	//Memory area where access error occured
  OB122_MEM_ADDR : WORD ;	//Memory address where access error occured
  OB122_BLK_NUM : WORD ;	//Block number in which error occured
  OB122_PRG_ADDR : WORD ;	//Program address where error occured
  OB122_DATE_TIME : DATE_AND_TIME ;	//Date and time OB1 started
END_VAR
BEGIN
// (block stored without names or comments; labels and parameter names are numbered)
END_ORGANIZATION_BLOCK
